(*
SPDX-FileCopyrightText: © 2026 Oleksandr Tiutyk <trofimich@gmail.com>
SPDX-License-Identifier: MIT
License: https://opensource.org/license/mit
*)

{attribute 'no_explicit_call' := 'do not call this function block directly'}
FUNCTION_BLOCK LogFilter EXTENDS TOF_Core.Object IMPLEMENTS TOF_Core.ILogFilter
VAR_STAT
	//! <summary>Class name shared by all instances of this function block.</summary>
	_ClassName : STRING := __POUNAME();
END_VAR

{attribute 'monitoring' := 'call'}
PROPERTY ClassName : REFERENCE TO STRING
GET
ClassName REF= _ClassName;
END_GET
END_PROPERTY

{attribute 'monitoring' := 'call'}
PROPERTY NamespaceName : REFERENCE TO STRING
GET
NamespaceName REF= CurrentNamespace.Name;
END_GET
END_PROPERTY

{attribute 'monitoring' := 'call'}
PROPERTY SelfSize : ULINT
GET
SelfSize := XSIZEOF(THIS^);
END_GET
END_PROPERTY

METHOD ShouldLog : BOOL
VAR_IN_OUT CONSTANT
	category : TOF_Core.LOG_CATEGORY;
	topics : ARRAY [*] OF WSTRING;		
END_VAR
VAR
	i : DINT;
	interestedTokenFound : BOOL;
END_VAR
IF category > TOF_Core.LOG_CATEGORY.WARNING THEN
	ShouldLog := TRUE;
	RETURN;
END_IF

FOR i := LOWER_BOUND(topics, 1) TO UPPER_BOUND(topics, 1) DO
	IF topics[i] = "Timer" THEN
		RETURN;		
	END_IF
	
	IF topics[i] = "Workflow" OR_ELSE topics[i] = "Activity" THEN
		interestedTokenFound := TRUE;
	END_IF
END_FOR

ShouldLog := interestedTokenFound;
END_METHOD

END_FUNCTION_BLOCK

(* stored: Version 1.1.0.1
   POU LogFilter: Id {cc064da6-60c8-4032-9142-fe9dba46e6ef}, SpecialFunc None
   Property ClassName: Id {e7368c67-1e3f-4813-b1e8-7c2a0ce72182}
   Get Get: Id {090000aa-ea3e-49d7-8f45-dc489acef136}
   Property NamespaceName: Id {a847b108-40a2-4d86-a5db-36e8c9e78a61}
   Get Get: Id {53931b67-135f-4aad-aa40-6834e70ccc21}
   Property SelfSize: Id {00e55284-03ff-4a61-bf71-455fd9c88c9d}
   Get Get: Id {62a15046-e257-4b70-9ef3-a8490f97cfdd}
   Method ShouldLog: Id {dea599ed-3dde-4aca-8d23-02d039b7c9b9} *)
